(* Logix 5000 project; controller SX_V040001_C001 vendor 1 type 14 code 77 rev 16.23; software revision 16.04; part 9 of 35 *)
(* tags used below, declared in another part *)
   ANA_OUTPUT_SIM : INT[8];
   CMD : INT[36];
   command_number : INT;
   command_value : INT;
   DB_A_IO : INT[16];
   DIGI_OUTPUT_SIM : DINT[3];
   DIGI_OUTPUT_SIM_REVERSE : DINT[3];
   G_AOutput : DINT[8];
   G_DOutput : DINT[3];
   m_on_off_line : BOOL;
   pointer_bcc_in : DINT;
   pointer_bcc_out : DINT;
   REMOTE_DATA_IN : INT[510];
   REMOTE_DATA_OUT : INT[510];
   temp_bcc_in : DINT;
   temp_bcc_out : DINT;
(* MainProgram, continued *)

ROUTINE CalcBCC_IN   (* ladder *)
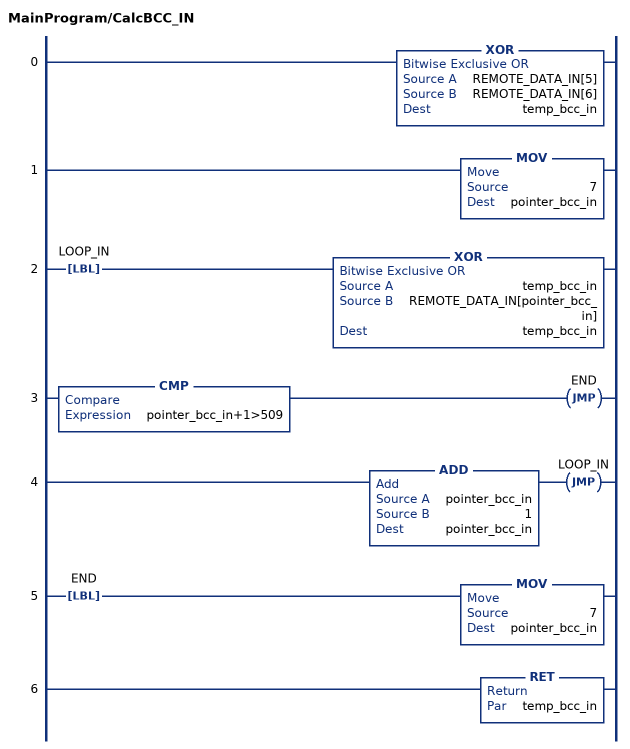
   0: XOR(REMOTE_DATA_IN[5],REMOTE_DATA_IN[6],temp_bcc_in);
   1: MOV(7,pointer_bcc_in);
   2: LBL(LOOP_IN)XOR(temp_bcc_in,REMOTE_DATA_IN[pointer_bcc_in],temp_bcc_in);
   3: CMP(pointer_bcc_in+1>509)JMP(END);
   4: ADD(pointer_bcc_in,1,pointer_bcc_in)JMP(LOOP_IN);
   5: LBL(END)MOV(7,pointer_bcc_in);
   6: RET(temp_bcc_in);
END_ROUTINE

ROUTINE CalcBCC_OUT   (* ladder *)
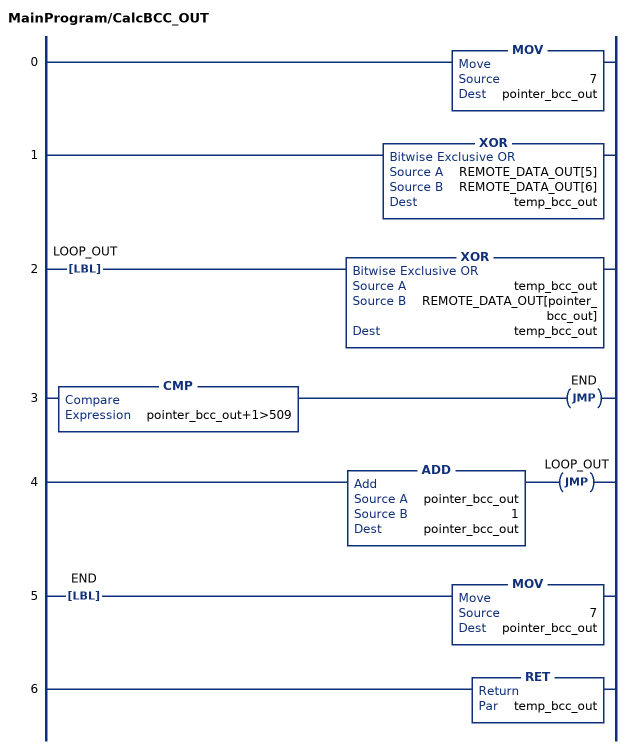
   0: MOV(7,pointer_bcc_out);
   1: XOR(REMOTE_DATA_OUT[5],REMOTE_DATA_OUT[6],temp_bcc_out);
   2: LBL(LOOP_OUT)XOR(temp_bcc_out,REMOTE_DATA_OUT[pointer_bcc_out],temp_bcc_out);
   3: CMP(pointer_bcc_out+1>509)JMP(END);
   4: ADD(pointer_bcc_out,1,pointer_bcc_out)JMP(LOOP_OUT);
   5: LBL(END)MOV(7,pointer_bcc_out);
   6: RET(temp_bcc_out);
END_ROUTINE

ROUTINE ComDeco_1   (* ladder *)
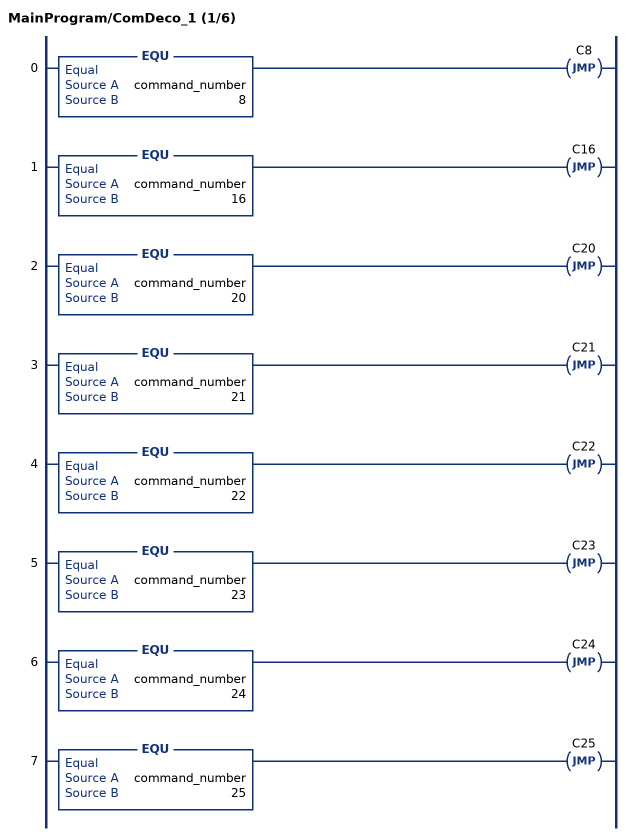
   0: EQU(command_number,8)JMP(C8);
   1: EQU(command_number,16)JMP(C16);
   2: EQU(command_number,20)JMP(C20);
   3: EQU(command_number,21)JMP(C21);
   4: EQU(command_number,22)JMP(C22);
   5: EQU(command_number,23)JMP(C23);
   6: EQU(command_number,24)JMP(C24);
   7: EQU(command_number,25)JMP(C25);
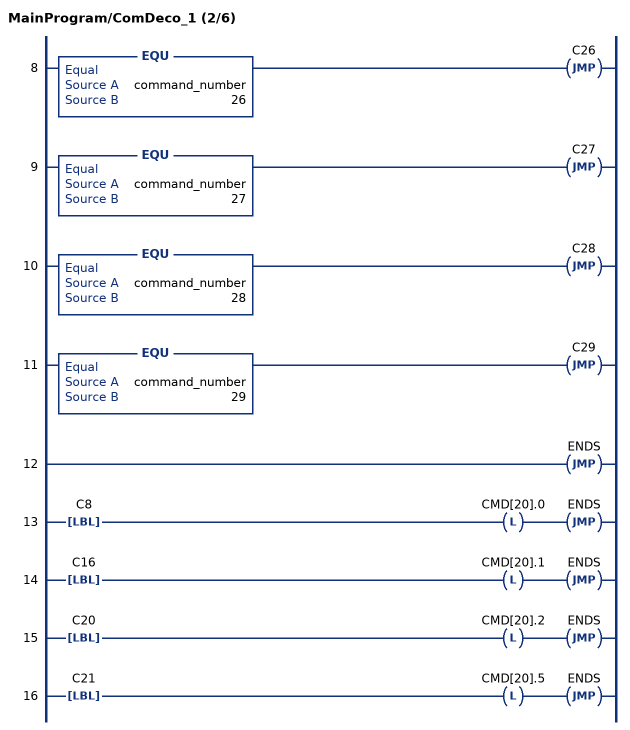
   8: EQU(command_number,26)JMP(C26);
   9: EQU(command_number,27)JMP(C27);
   10: EQU(command_number,28)JMP(C28);
   11: EQU(command_number,29)JMP(C29);
   12: JMP(ENDS);
   13: LBL(C8)OTL(CMD[20].0)JMP(ENDS);
   14: LBL(C16)OTL(CMD[20].1)JMP(ENDS);
   15: LBL(C20)OTL(CMD[20].2)JMP(ENDS);
   16: LBL(C21)OTL(CMD[20].5)JMP(ENDS);
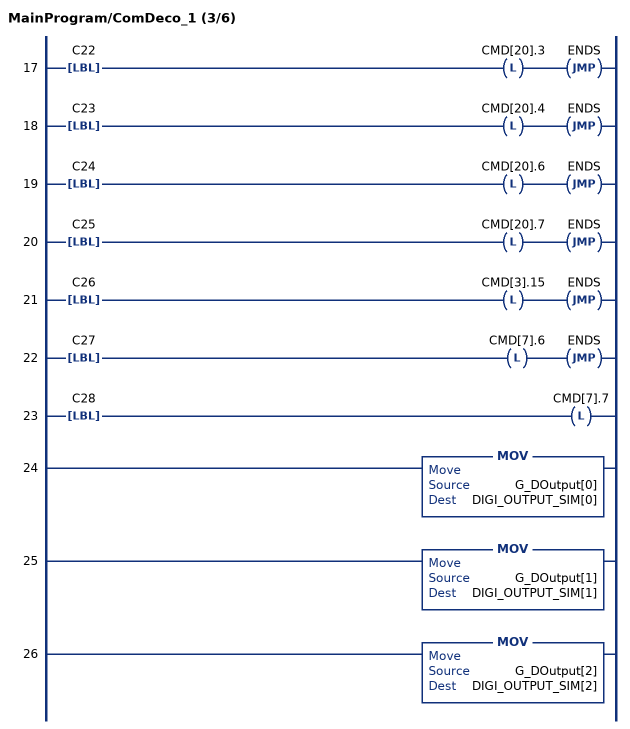
   17: LBL(C22)OTL(CMD[20].3)JMP(ENDS);
   18: LBL(C23)OTL(CMD[20].4)JMP(ENDS);
   19: LBL(C24)OTL(CMD[20].6)JMP(ENDS);
   20: LBL(C25)OTL(CMD[20].7)JMP(ENDS);
   21: LBL(C26)OTL(CMD[3].15)JMP(ENDS);
   22: LBL(C27)OTL(CMD[7].6)JMP(ENDS);
   23: LBL(C28)OTL(CMD[7].7);
   24: MOV(G_DOutput[0],DIGI_OUTPUT_SIM[0]);
   25: MOV(G_DOutput[1],DIGI_OUTPUT_SIM[1]);
   26: MOV(G_DOutput[2],DIGI_OUTPUT_SIM[2]);
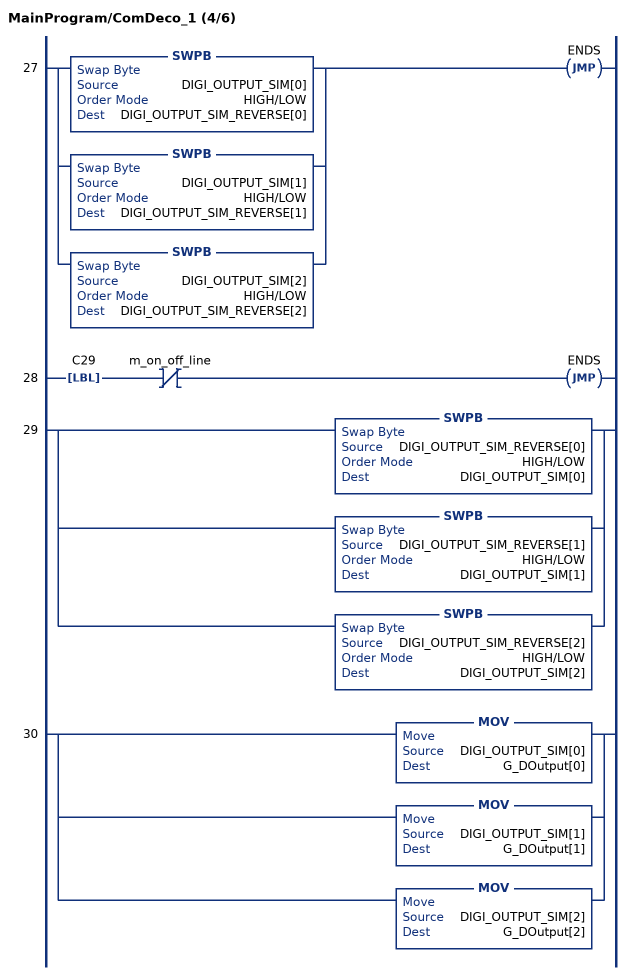
   27: [SWPB(DIGI_OUTPUT_SIM[0],HIGH/LOW,DIGI_OUTPUT_SIM_REVERSE[0]) ,SWPB(DIGI_OUTPUT_SIM[1],HIGH/LOW,DIGI_OUTPUT_SIM_REVERSE[1]) ,SWPB(DIGI_OUTPUT_SIM[2],HIGH/LOW,DIGI_OUTPUT_SIM_REVERSE[2]) ]JMP(ENDS);
   28: LBL(C29)XIO(m_on_off_line)JMP(ENDS);
   29: [SWPB(DIGI_OUTPUT_SIM_REVERSE[0],HIGH/LOW,DIGI_OUTPUT_SIM[0]) ,SWPB(DIGI_OUTPUT_SIM_REVERSE[1],HIGH/LOW,DIGI_OUTPUT_SIM[1]) ,SWPB(DIGI_OUTPUT_SIM_REVERSE[2],HIGH/LOW,DIGI_OUTPUT_SIM[2]) ];
   30: [MOV(DIGI_OUTPUT_SIM[0],G_DOutput[0]) ,MOV(DIGI_OUTPUT_SIM[1],G_DOutput[1]) ,MOV(DIGI_OUTPUT_SIM[2],G_DOutput[2]) ];
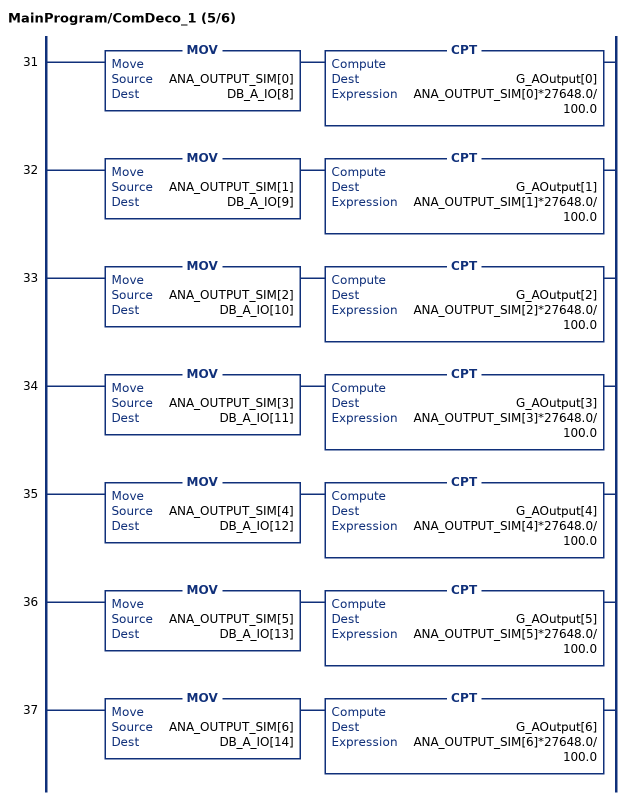
   31: MOV(ANA_OUTPUT_SIM[0],DB_A_IO[8])CPT(G_AOutput[0],ANA_OUTPUT_SIM[0]*27648.0/100.0);
   32: MOV(ANA_OUTPUT_SIM[1],DB_A_IO[9])CPT(G_AOutput[1],ANA_OUTPUT_SIM[1]*27648.0/100.0);
   33: MOV(ANA_OUTPUT_SIM[2],DB_A_IO[10])CPT(G_AOutput[2],ANA_OUTPUT_SIM[2]*27648.0/100.0);
   34: MOV(ANA_OUTPUT_SIM[3],DB_A_IO[11])CPT(G_AOutput[3],ANA_OUTPUT_SIM[3]*27648.0/100.0);
   35: MOV(ANA_OUTPUT_SIM[4],DB_A_IO[12])CPT(G_AOutput[4],ANA_OUTPUT_SIM[4]*27648.0/100.0);
   36: MOV(ANA_OUTPUT_SIM[5],DB_A_IO[13])CPT(G_AOutput[5],ANA_OUTPUT_SIM[5]*27648.0/100.0);
   37: MOV(ANA_OUTPUT_SIM[6],DB_A_IO[14])CPT(G_AOutput[6],ANA_OUTPUT_SIM[6]*27648.0/100.0);
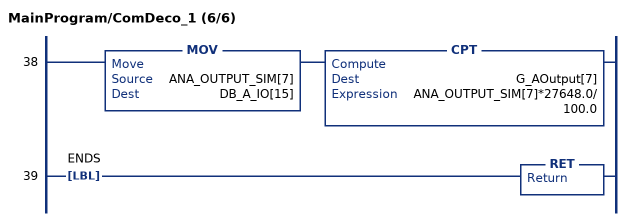
   38: MOV(ANA_OUTPUT_SIM[7],DB_A_IO[15])CPT(G_AOutput[7],ANA_OUTPUT_SIM[7]*27648.0/100.0);
   39: LBL(ENDS)RET();
END_ROUTINE

ROUTINE ComDeco_2   (* ladder *)
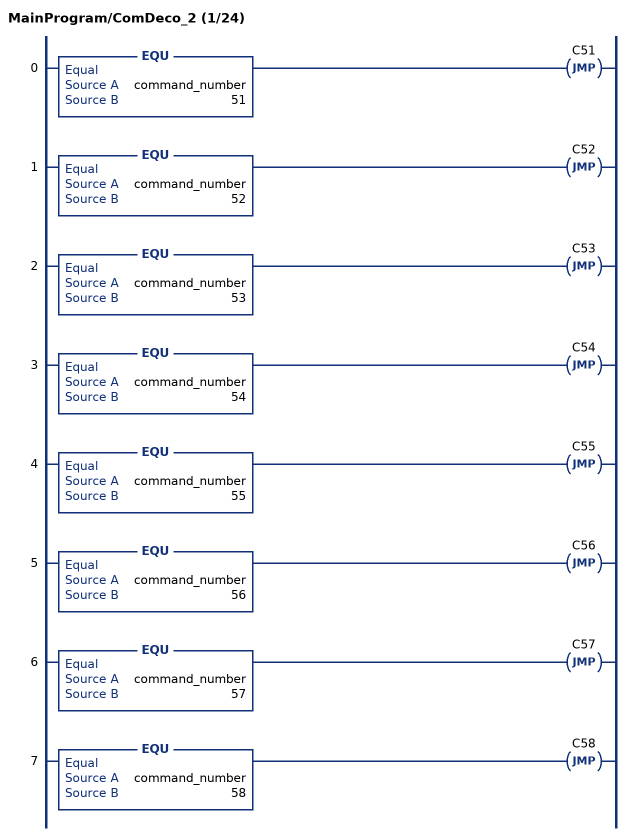
   0: EQU(command_number,51)JMP(C51);
   1: EQU(command_number,52)JMP(C52);
   2: EQU(command_number,53)JMP(C53);
   3: EQU(command_number,54)JMP(C54);
   4: EQU(command_number,55)JMP(C55);
   5: EQU(command_number,56)JMP(C56);
   6: EQU(command_number,57)JMP(C57);
   7: EQU(command_number,58)JMP(C58);
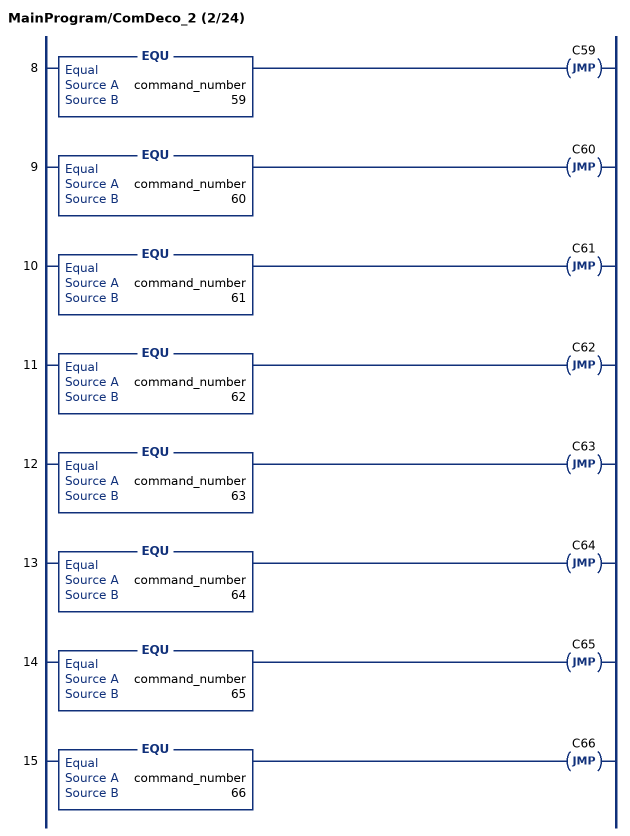
   8: EQU(command_number,59)JMP(C59);
   9: EQU(command_number,60)JMP(C60);
   10: EQU(command_number,61)JMP(C61);
   11: EQU(command_number,62)JMP(C62);
   12: EQU(command_number,63)JMP(C63);
   13: EQU(command_number,64)JMP(C64);
   14: EQU(command_number,65)JMP(C65);
   15: EQU(command_number,66)JMP(C66);
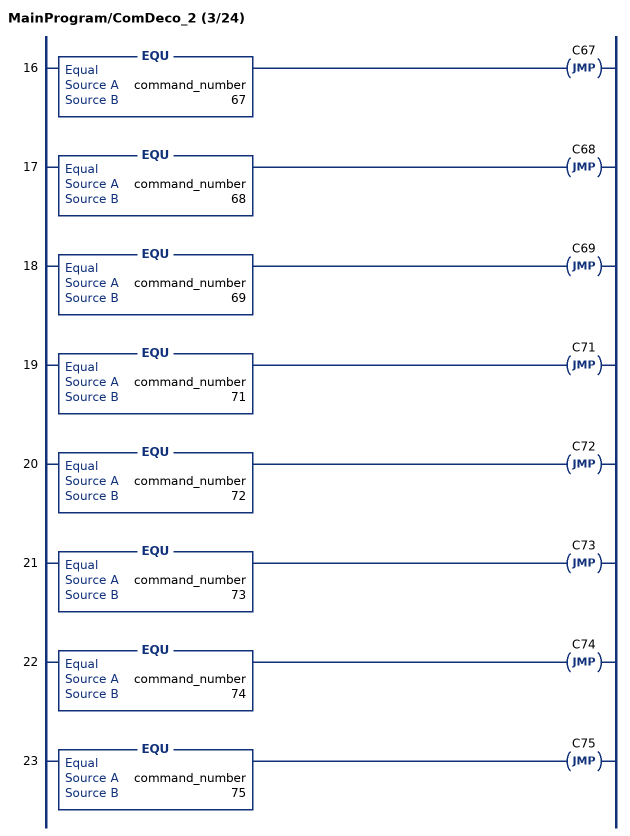
   16: EQU(command_number,67)JMP(C67);
   17: EQU(command_number,68)JMP(C68);
   18: EQU(command_number,69)JMP(C69);
   19: EQU(command_number,71)JMP(C71);
   20: EQU(command_number,72)JMP(C72);
   21: EQU(command_number,73)JMP(C73);
   22: EQU(command_number,74)JMP(C74);
   23: EQU(command_number,75)JMP(C75);
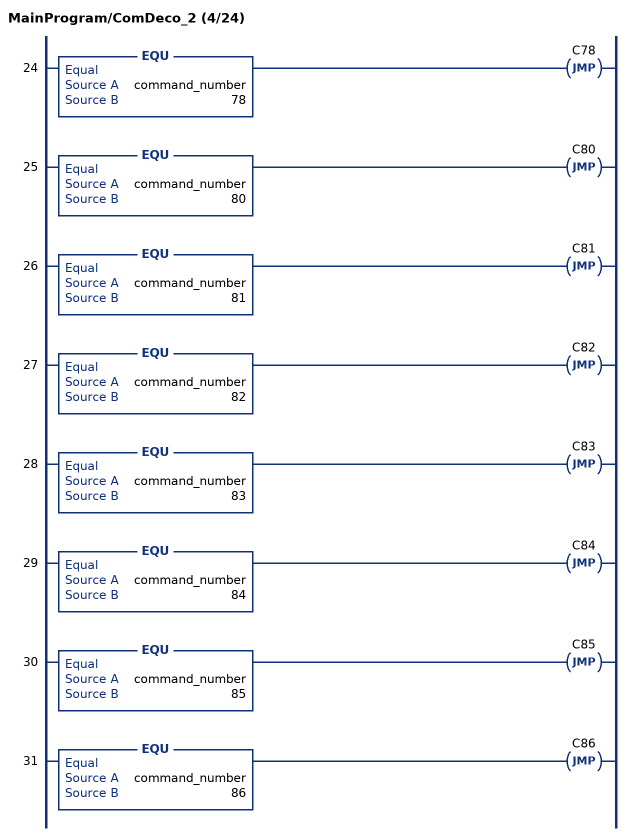
   24: EQU(command_number,78)JMP(C78);
   25: EQU(command_number,80)JMP(C80);
   26: EQU(command_number,81)JMP(C81);
   27: EQU(command_number,82)JMP(C82);
   28: EQU(command_number,83)JMP(C83);
   29: EQU(command_number,84)JMP(C84);
   30: EQU(command_number,85)JMP(C85);
   31: EQU(command_number,86)JMP(C86);
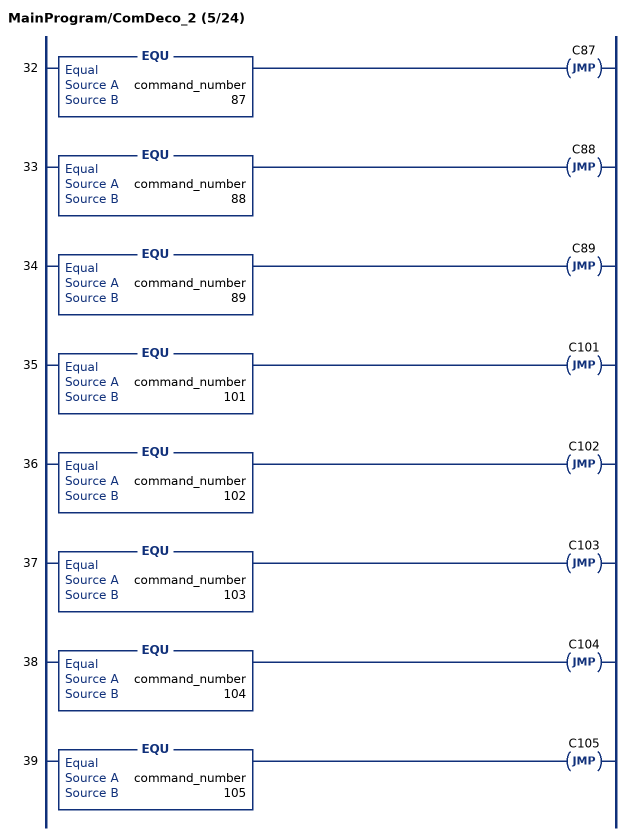
   32: EQU(command_number,87)JMP(C87);
   33: EQU(command_number,88)JMP(C88);
   34: EQU(command_number,89)JMP(C89);
   35: EQU(command_number,101)JMP(C101);
   36: EQU(command_number,102)JMP(C102);
   37: EQU(command_number,103)JMP(C103);
   38: EQU(command_number,104)JMP(C104);
   39: EQU(command_number,105)JMP(C105);
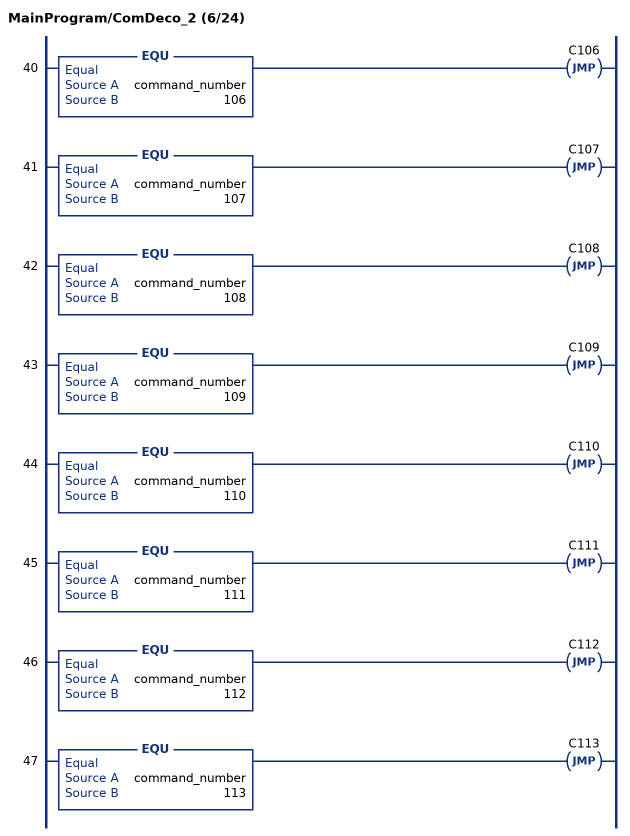
   40: EQU(command_number,106)JMP(C106);
   41: EQU(command_number,107)JMP(C107);
   42: EQU(command_number,108)JMP(C108);
   43: EQU(command_number,109)JMP(C109);
   44: EQU(command_number,110)JMP(C110);
   45: EQU(command_number,111)JMP(C111);
   46: EQU(command_number,112)JMP(C112);
   47: EQU(command_number,113)JMP(C113);
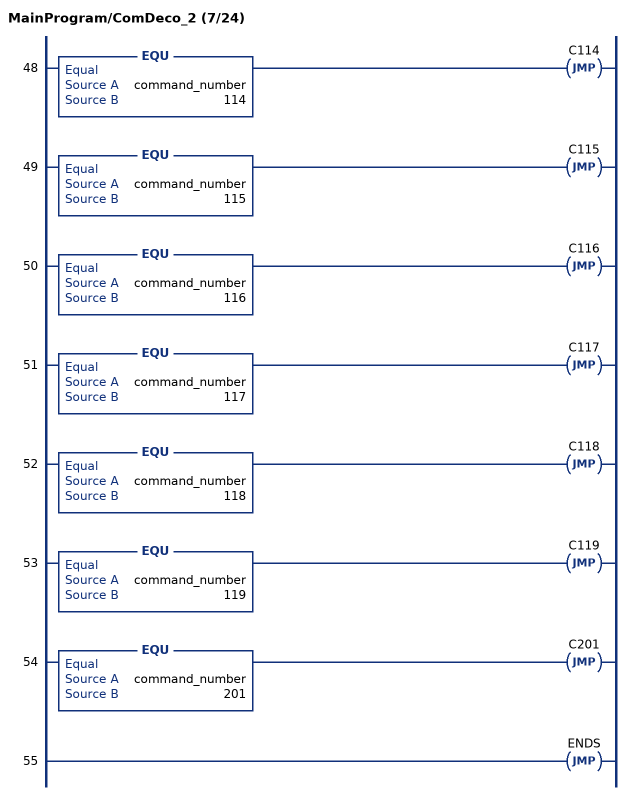
   48: EQU(command_number,114)JMP(C114);
   49: EQU(command_number,115)JMP(C115);
   50: EQU(command_number,116)JMP(C116);
   51: EQU(command_number,117)JMP(C117);
   52: EQU(command_number,118)JMP(C118);
   53: EQU(command_number,119)JMP(C119);
   54: EQU(command_number,201)JMP(C201);
   55: JMP(ENDS);
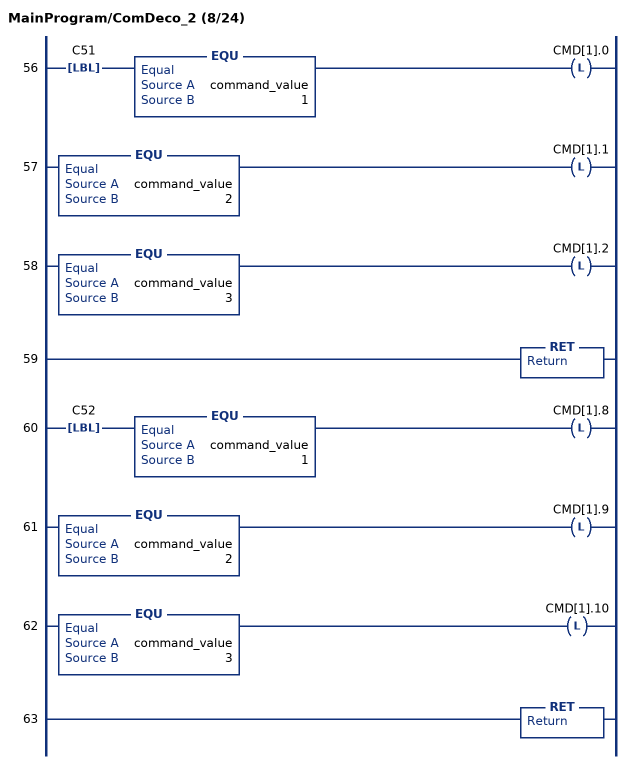
   56: LBL(C51)EQU(command_value,1)OTL(CMD[1].0);
   57: EQU(command_value,2)OTL(CMD[1].1);
   58: EQU(command_value,3)OTL(CMD[1].2);
   59: RET();
   60: LBL(C52)EQU(command_value,1)OTL(CMD[1].8);
   61: EQU(command_value,2)OTL(CMD[1].9);
   62: EQU(command_value,3)OTL(CMD[1].10);
   63: RET();
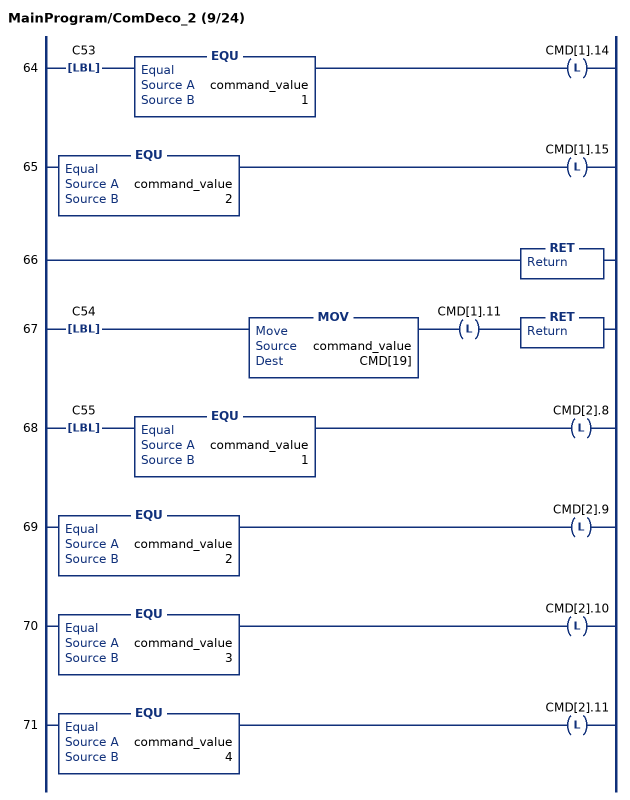
   64: LBL(C53)EQU(command_value,1)OTL(CMD[1].14);
   65: EQU(command_value,2)OTL(CMD[1].15);
   66: RET();
   67: LBL(C54)MOV(command_value,CMD[19])OTL(CMD[1].11)RET();
   68: LBL(C55)EQU(command_value,1)OTL(CMD[2].8);
   69: EQU(command_value,2)OTL(CMD[2].9);
   70: EQU(command_value,3)OTL(CMD[2].10);
   71: EQU(command_value,4)OTL(CMD[2].11);
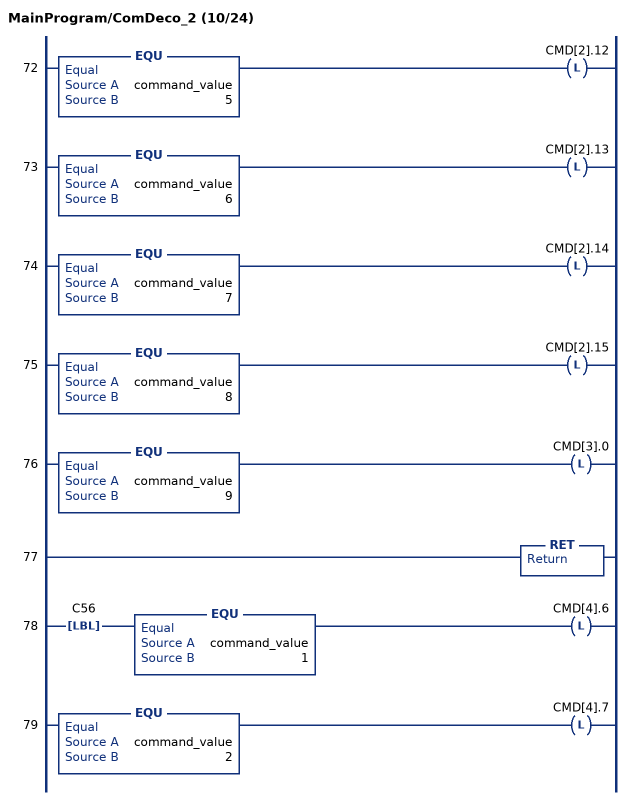
   72: EQU(command_value,5)OTL(CMD[2].12);
   73: EQU(command_value,6)OTL(CMD[2].13);
   74: EQU(command_value,7)OTL(CMD[2].14);
   75: EQU(command_value,8)OTL(CMD[2].15);
   76: EQU(command_value,9)OTL(CMD[3].0);
   77: RET();
   78: LBL(C56)EQU(command_value,1)OTL(CMD[4].6);
   79: EQU(command_value,2)OTL(CMD[4].7);
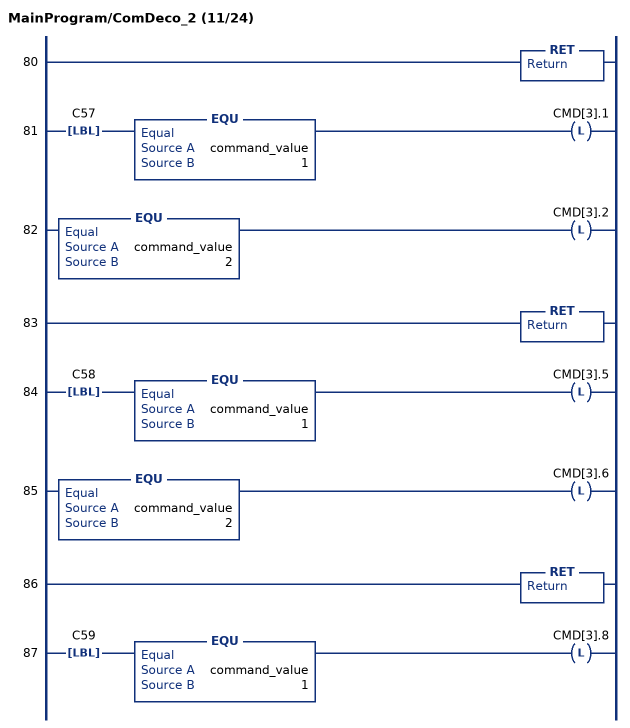
   80: RET();
   81: LBL(C57)EQU(command_value,1)OTL(CMD[3].1);
   82: EQU(command_value,2)OTL(CMD[3].2);
   83: RET();
   84: LBL(C58)EQU(command_value,1)OTL(CMD[3].5);
   85: EQU(command_value,2)OTL(CMD[3].6);
   86: RET();
   87: LBL(C59)EQU(command_value,1)OTL(CMD[3].8);
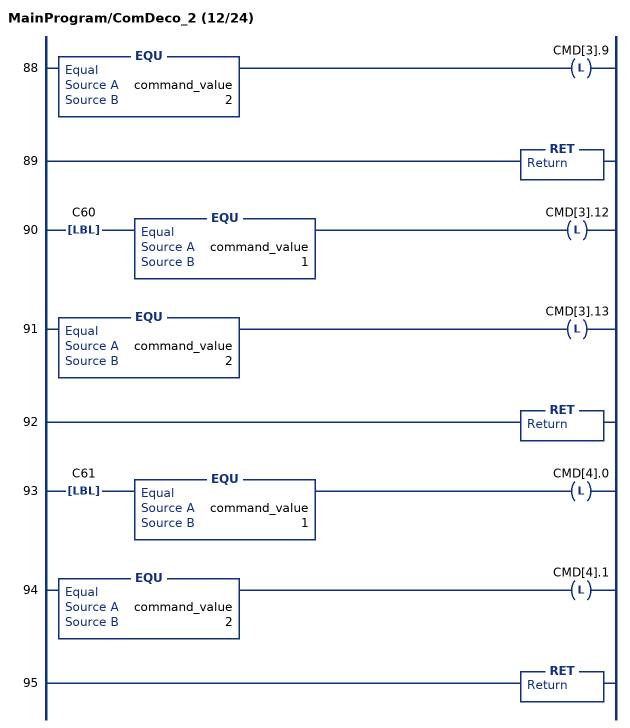
   88: EQU(command_value,2)OTL(CMD[3].9);
   89: RET();
   90: LBL(C60)EQU(command_value,1)OTL(CMD[3].12);
   91: EQU(command_value,2)OTL(CMD[3].13);
   92: RET();
   93: LBL(C61)EQU(command_value,1)OTL(CMD[4].0);
   94: EQU(command_value,2)OTL(CMD[4].1);
   95: RET();
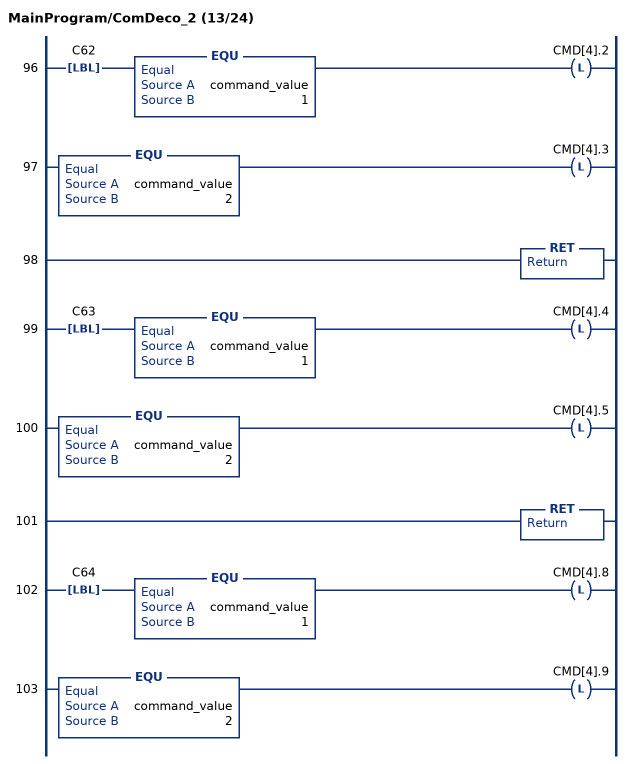
   96: LBL(C62)EQU(command_value,1)OTL(CMD[4].2);
   97: EQU(command_value,2)OTL(CMD[4].3);
   98: RET();
   99: LBL(C63)EQU(command_value,1)OTL(CMD[4].4);
   100: EQU(command_value,2)OTL(CMD[4].5);
   101: RET();
   102: LBL(C64)EQU(command_value,1)OTL(CMD[4].8);
   103: EQU(command_value,2)OTL(CMD[4].9);
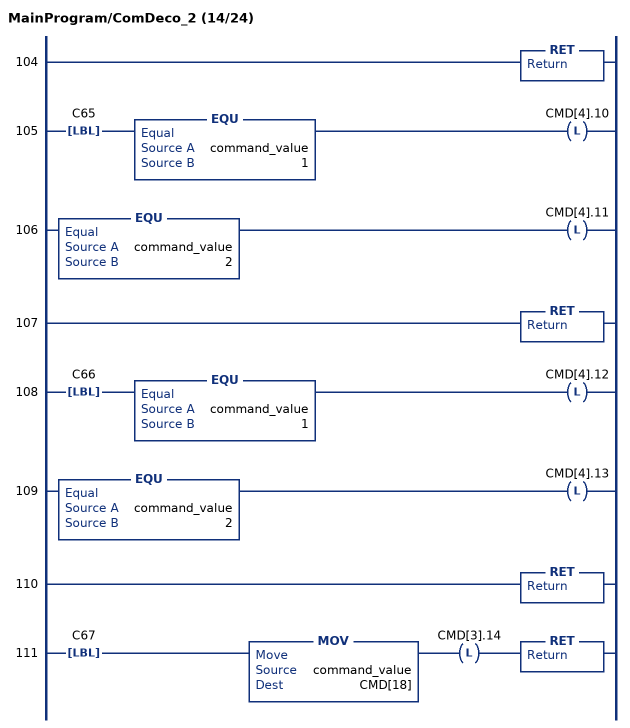
   104: RET();
   105: LBL(C65)EQU(command_value,1)OTL(CMD[4].10);
   106: EQU(command_value,2)OTL(CMD[4].11);
   107: RET();
   108: LBL(C66)EQU(command_value,1)OTL(CMD[4].12);
   109: EQU(command_value,2)OTL(CMD[4].13);
   110: RET();
   111: LBL(C67)MOV(command_value,CMD[18])OTL(CMD[3].14)RET();
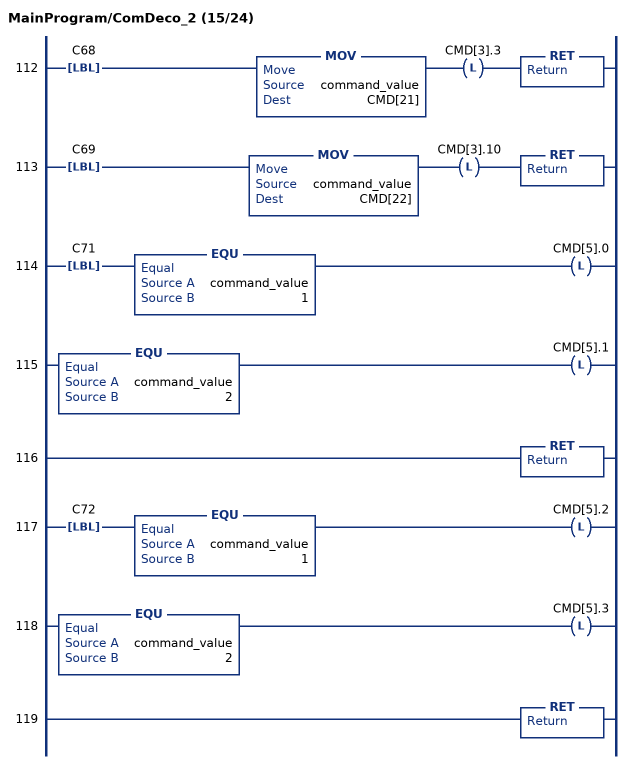
   112: LBL(C68)MOV(command_value,CMD[21])OTL(CMD[3].3)RET();
   113: LBL(C69)MOV(command_value,CMD[22])OTL(CMD[3].10)RET();
   114: LBL(C71)EQU(command_value,1)OTL(CMD[5].0);
   115: EQU(command_value,2)OTL(CMD[5].1);
   116: RET();
   117: LBL(C72)EQU(command_value,1)OTL(CMD[5].2);
   118: EQU(command_value,2)OTL(CMD[5].3);
   119: RET();
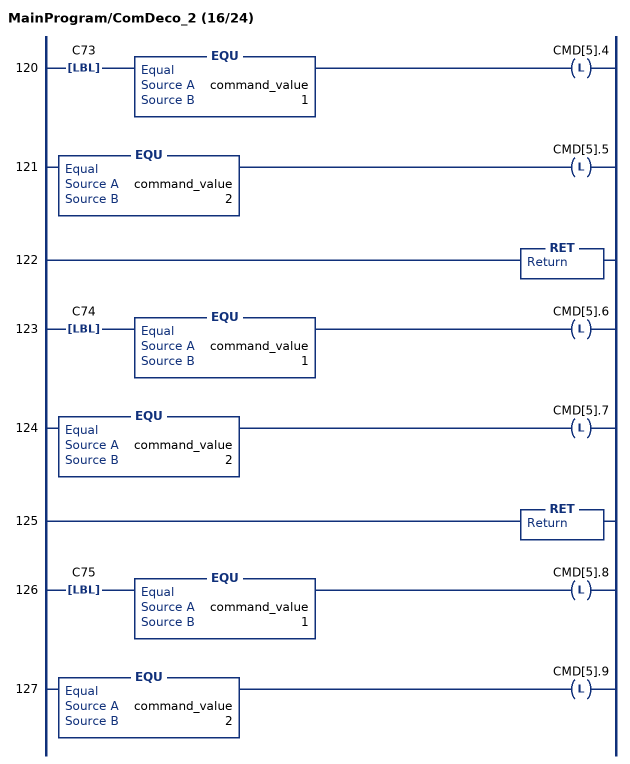
   120: LBL(C73)EQU(command_value,1)OTL(CMD[5].4);
   121: EQU(command_value,2)OTL(CMD[5].5);
   122: RET();
   123: LBL(C74)EQU(command_value,1)OTL(CMD[5].6);
   124: EQU(command_value,2)OTL(CMD[5].7);
   125: RET();
   126: LBL(C75)EQU(command_value,1)OTL(CMD[5].8);
   127: EQU(command_value,2)OTL(CMD[5].9);
